// Mitsubishi GX Works2 project: mcode   PLC: Q02/Q02H

PROGRAM MAIN
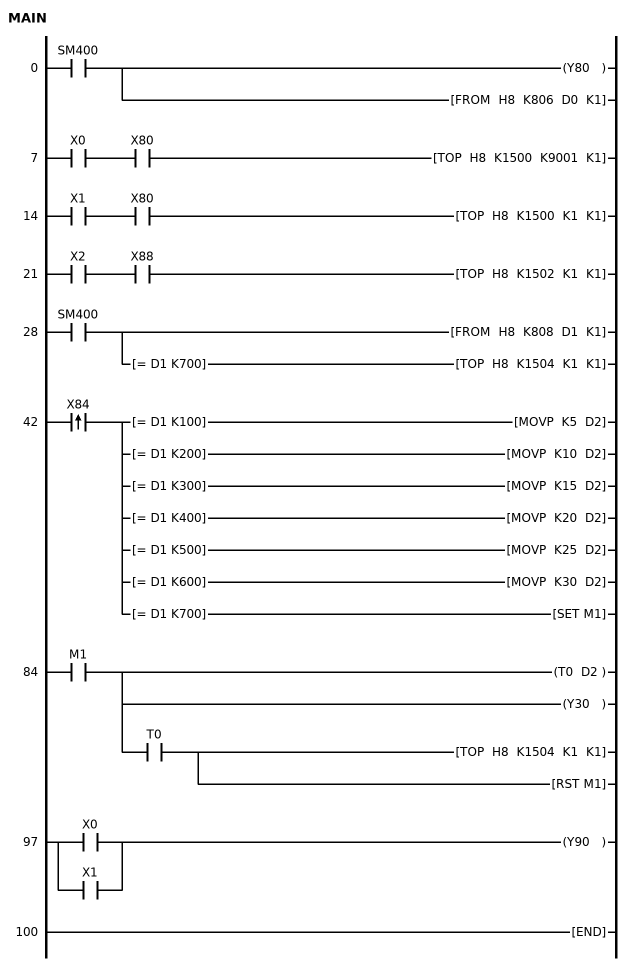
0     LD      SM400
      OUT     Y80
      FROM    H8 K806 D0 K1
7     LD      X0
      AND     X80
      TOP     H8 K1500 K9001 K1
14    LD      X1
      AND     X80
      TOP     H8 K1500 K1 K1
21    LD      X2
      AND     X88
      TOP     H8 K1502 K1 K1
28    LD      SM400
      FROM    H8 K808 D1 K1
      AND=    D1 K700
      TOP     H8 K1504 K1 K1
42    LDP     X84
      MPS
      AND=    D1 K100
      MOVP    K5 D2
      MRD
      AND=    D1 K200
      MOVP    K10 D2
      MRD
      AND=    D1 K300
      MOVP    K15 D2
      MRD
      AND=    D1 K400
      MOVP    K20 D2
      MRD
      AND=    D1 K500
      MOVP    K25 D2
      MRD
      AND=    D1 K600
      MOVP    K30 D2
      MPP
      AND=    D1 K700
      SET     M1
84    LD      M1
      OUT     T0 D2
      OUT     Y30
      AND     T0
      TOP     H8 K1504 K1 K1
      RST     M1
97    LD      X0
      OR      X1
      OUT     Y90
100   END
END_PROGRAM
